TYPE ST_ProgramListStruct :
STRUCT
	ID: LINT;
	Name: STRING(255);
END_STRUCT
END_TYPE

(* stored: Version 1.1.0.1, ProductVersion 3.1.4022.12
   DUT ST_ProgramListStruct: Id {168479d3-bc29-4477-8f61-7d998dd7298f} *)
